// Mitsubishi GX Works2 project: ATIVIDADE VERSIONAMENTO   PLC: Q03UDV

PROGRAM MAIN
VAR
  SAIDA : BOOL;
END_VAR
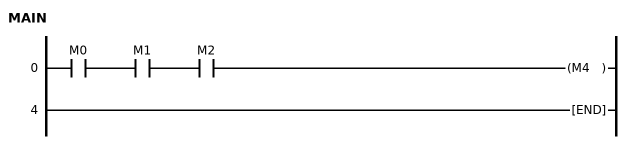
0     LD      M0
      AND     M1
      AND     M2
      OUT     M4
4     END
END_PROGRAM
